{attribute 'GeneratedUsingTerminal: EL3356-0030-0025'}
{attribute addProperty BoxType "EL3356-0030-0025"}
{attribute addProperty Id "ValueAT %I*DINT4"}
{attribute addProperty CRC "3910704203"}
{attribute addProperty Size "4"}
TYPE RMB_Value_INT_E9189C4B :
STRUCT
	{attribute addProperty Name "Value"}
	Value AT %I* : DINT;
END_STRUCT
END_TYPE

(* stored: Version 1.2.0.0, ProductVersion 3.1.4024.9
   DUT RMB_Value_INT_E9189C4B: Id {0afd2f0d-fa19-4429-8a6d-574466d3e2aa} *)
